DEVICE_TYPE TEST_DEVICE (* Minimal device type for mapping tests *)
  (* Standard: 61499-1 *)
  (* Version 1.0, 2026-02-23, test, 4diac tests *)
  VAR_INPUT
    MGR_ID : WSTRING := "localhost:61499"; (* Device manager socket ID *)
  END_VAR
END_DEVICE_TYPE
